// TIA Portal V16 export
// export: Created 2022-11-17T11:55:36.6386521Z, ExportSetting WithDefaults, DisplayName Totally Integrated Automation Portal, DisplayVersion V16 Update 6, DisplayName TIA Portal Version Control Interface, DisplayVersion V16 Update 2, DisplayName TIA Portal Openness, DisplayVersion V16 Update 6, DisplayName SINAMICS Startdrive Advanced, DisplayVersion V16 Update 5, DisplayName SINAMICS Startdrive G130, G150, S120, S150, SINAMICS MV, S210, DisplayVersion V16 Update 5, DisplayName SINAMICS Startdrive G110M, G120, G120C, G120D, G120P, G115D, DisplayVersion V16 Update 5, DisplayName STEP 7 Professional, DisplayVersion V16 Update 6, DisplayName STEP 7 Safety, DisplayVersion V16, DisplayName WinCC Advanced, DisplayVersion V16 Update 6
DATA_BLOCK "DB321_PID_M20"   // DB321
TITLE = PID
{ S7_Optimized_Access := 'FALSE' }
VERSION : 0.1
// stored: AutoNumber false, IsOnlyStoredInLoadMemory false, IsWriteProtectedInAS false
   VAR RETAIN
      PID { S7_SetPoint := 'True'} : "M20";
   END_VAR
BEGIN
   PID.M20_P00 := 0;
   PID.M20_P01 := 70;
   PID.M20_P02 := 15;
   PID.M20_P03 := 0;
   PID.M20_P04 := 60;
   PID.M20_P05 := 7;
   PID.M20_P06 := 200;
   PID.M20_P07 := 200;
   PID.M20_P08 := 65;
   PID.M20_P09 := 240;
   PID.M20_P10 := 100;
   PID.M20_P11 := 128;
   PID.M20_P12 := 10;
   PID.M20_P13 := 0;
   PID.M20_P14 := 6;
   PID.M20_P15 := 50;
   PID.M20_P20 := 0;
   PID.M20_P21 := 0;
   PID.M20_P22 := 0;
   PID.M20_P23 := 0;
   PID.M20_P24 := 0;
   PID.M20_P25 := 0;
END_DATA_BLOCK
